Universal Robots PolyScope program: partmover03_touch.urp

Program partmover03_touch (installation=default directory=/programs createdIn=5.9.1.1031110 lastSavedIn=5.9.1.1031110 robotSerialNumber=20195501059)
Calibrated DH parameters: a=[0.000146, -0.418764, -0.053981, 0.000058, -0.000023, 0]; d=[0.162545, 37.319448, -206.067439, 168.881546, 0.09955, 0.099464]; alpha=[1.57004, -0.001979, 0.002304, 1.570607, -1.57066, 0]; deltaTheta=[0, -0.174616, -1.258233, 1.432844, -0.000001, 0]
InitVariablesNode variables(variable(name=seek_v, expression=20))
BeforeStart
  seek_v := seek_v
  URCap Gripper Activate (Robotiq_Grippers, Robotiq Inc.) dataModel(ResetAndActivateKey=false)
Robot Program (runOnlyOnce=false)
  Call Pick1
  Call Place2
  Call Pick2
  Call Place1
SubProgram -> Pick1
SubProgram -> Place2
SubProgram -> Pick2
SubProgram -> Place1
SubProgram Pick1 (keepSynchronizedWithDisk=false)
  MoveL speed 250 mm/s, acceleration 1200 mm/s^2 (useActiveTCP=true) feature=Base
    Waypoint approach1: TCP in base x=233.098 y=-416.683 z=53.907 mm, rx=-2.1706 ry=-2.2616 rz=-0.0123 rad; joints [102.865, -81.519, 121.946, -129.844, 270.216, 100.549] deg; TCP offset x=0 y=0 z=174 mm, rx=0 ry=0 rz=0 rad
    URCap Gripper (Robotiq_Grippers, Robotiq Inc.) dataModel(position=100.0, force=100.0, speed=100.0, positionInDouble=100.0, forceInDouble=100.0, speedInDouble=100.0, slaveIds=[9], blocking=true)
    MoveDirectionNode (selectedDirection=ZPlus toolParams=0.02, 0.5) feature=Joint_6_name
      Until TOOL_CONTACT_DETECTION (allowActions=false retraction=0.003 decelerationAcceleration=1 decelerationAngularAcceleration=34.906585)
    URCap Gripper (Robotiq_Grippers, Robotiq Inc.) dataModel(position=40.0, force=100.0, speed=100.0, positionInDouble=40.0, forceInDouble=100.0, speedInDouble=100.0, slaveIds=[9], blocking=true)
    MoveDirectionNode (selectedDirection=ZPlus) feature=Joint_6_name
      Until DISTANCE (allowActions=false deceleration=3 distanceNodeType=STOP) Distance=0.015; motionParameters(blendRadius=0)
    URCap Gripper (Robotiq_Grippers, Robotiq Inc.) dataModel(position=100.0, force=100.0, speed=100.0, positionInDouble=100.0, forceInDouble=100.0, speedInDouble=100.0, slaveIds=[9], blocking=true)
    Waypoint approach1: TCP in base x=233.098 y=-416.683 z=53.907 mm, rx=-2.1706 ry=-2.2616 rz=-0.0123 rad; joints [102.865, -81.519, 121.946, -129.844, 270.216, 100.549] deg
SubProgram Place2 (keepSynchronizedWithDisk=false)
  MoveL speed 250 mm/s, acceleration 1200 mm/s^2 (useActiveTCP=true) feature=Base
    Waypoint approach2: TCP in base x=356.173 y=-318.335 z=53.911 mm, rx=-2.1706 ry=-2.2615 rz=-0.0123 rad; joints [121.755, -81.551, 122.012, -129.959, 270.395, 119.439] deg
    MoveDirectionNode (selectedDirection=ZPlus toolParams=0.02, 0.5) feature=Joint_6_name
      Until TOOL_CONTACT_DETECTION (allowActions=false retraction=0.001 decelerationAcceleration=1 decelerationAngularAcceleration=34.906585)
    URCap Gripper (Robotiq_Grippers, Robotiq Inc.) dataModel(position=40.0, force=100.0, speed=100.0, positionInDouble=40.0, forceInDouble=100.0, speedInDouble=100.0, slaveIds=[9], blocking=true)
    Waypoint approach2: TCP in base x=356.173 y=-318.335 z=53.911 mm, rx=-2.1706 ry=-2.2615 rz=-0.0123 rad; joints [121.755, -81.551, 122.012, -129.959, 270.395, 119.439] deg
SubProgram Pick2 (keepSynchronizedWithDisk=false)
  MoveL speed 250 mm/s, acceleration 1200 mm/s^2 (useActiveTCP=true) feature=Base
    Waypoint approach2: TCP in base x=356.173 y=-318.335 z=53.911 mm, rx=-2.1706 ry=-2.2615 rz=-0.0123 rad; joints [121.755, -81.551, 122.012, -129.959, 270.395, 119.439] deg
    URCap Gripper (Robotiq_Grippers, Robotiq Inc.) dataModel(position=100.0, force=100.0, speed=100.0, positionInDouble=100.0, forceInDouble=100.0, speedInDouble=100.0, slaveIds=[9], blocking=true)
    MoveDirectionNode (selectedDirection=ZPlus toolParams=0.02, 0.5) feature=Joint_6_name
      Until TOOL_CONTACT_DETECTION (allowActions=false retraction=0.003 decelerationAcceleration=1 decelerationAngularAcceleration=34.906585)
    URCap Gripper (Robotiq_Grippers, Robotiq Inc.) dataModel(position=40.0, force=100.0, speed=100.0, positionInDouble=40.0, forceInDouble=100.0, speedInDouble=100.0, slaveIds=[9], blocking=true)
    MoveDirectionNode (selectedDirection=ZPlus) feature=Joint_6_name
      Until DISTANCE (allowActions=false deceleration=3 distanceNodeType=STOP) Distance=0.015; motionParameters(blendRadius=0)
    URCap Gripper (Robotiq_Grippers, Robotiq Inc.) dataModel(position=100.0, force=100.0, speed=100.0, positionInDouble=100.0, forceInDouble=100.0, speedInDouble=100.0, slaveIds=[9], blocking=true)
    Waypoint approach2: TCP in base x=356.173 y=-318.335 z=53.911 mm, rx=-2.1706 ry=-2.2615 rz=-0.0123 rad; joints [121.755, -81.551, 122.012, -129.959, 270.395, 119.439] deg
SubProgram Place1 (keepSynchronizedWithDisk=false)
  MoveL speed 250 mm/s, acceleration 1200 mm/s^2 (useActiveTCP=true) feature=Base
    Waypoint approach1: TCP in base x=233.098 y=-416.683 z=53.907 mm, rx=-2.1706 ry=-2.2616 rz=-0.0123 rad; joints [102.865, -81.519, 121.946, -129.844, 270.216, 100.549] deg
    MoveDirectionNode (selectedDirection=ZPlus toolParams=0.02, 0.5) feature=Joint_6_name
      Until TOOL_CONTACT_DETECTION (allowActions=false retraction=0.001 decelerationAcceleration=1 decelerationAngularAcceleration=34.906585)
    URCap Gripper (Robotiq_Grippers, Robotiq Inc.) dataModel(position=40.0, force=100.0, speed=100.0, positionInDouble=40.0, forceInDouble=100.0, speedInDouble=100.0, slaveIds=[9], blocking=true)
    Waypoint approach1: TCP in base x=233.098 y=-416.683 z=53.907 mm, rx=-2.1706 ry=-2.2616 rz=-0.0123 rad; joints [102.865, -81.519, 121.946, -129.844, 270.216, 100.549] deg
